FUNCTION_BLOCK ABSTRACT KeyValueCollectionEventHandler EXTENDS MockEventHandler
VAR
	expectedOriginator : I_KeyValueCollection;
END_VAR

METHOD FB_init : BOOL
VAR_INPUT
	bInitRetains : BOOL; // if TRUE, the retain variables are initialized (warm start / cold start)
	bInCopyCode : BOOL;  // if TRUE, the instance afterwards gets moved into the copy code (online change)
	ExpectedOriginator : I_KeyValueCollection;
END_VAR
SetExpectedOriginator(ExpectedOriginator);
END_METHOD

METHOD PUBLIC SetExpectedOriginator
VAR_INPUT
	ExpectedOriginator : I_KeyValueCollection;
END_VAR
THIS^.expectedOriginator := ExpectedOriginator;
END_METHOD

END_FUNCTION_BLOCK

(* stored: Version 1.1.0.1, ProductVersion 3.1.4024.12
   POU KeyValueCollectionEventHandler: Id {a9f0bbbb-2b6d-4d8e-b52b-0c1f246b65c0}, SpecialFunc None
   Folder Constructor: Id {24ecd817-bcc7-42d3-9272-2b260fa45a63}
   Method FB_init: Id {f575aed3-b482-4dec-9702-1eb4dfb97ab2}
   Method SetExpectedOriginator: Id {d2eb46a6-1e61-4fd5-8a93-9f167c3261a9} *)
